FUNCTION_BLOCK FB_Cylinder IMPLEMENTS I_Cylinder
VAR_INPUT
	id	: INT;
END_VAR
VAR_OUTPUT
END_VAR
VAR
	bAtExtend 		AT %I*	: BOOL;
	bAtRetract 		AT %I*	: BOOL;
	bAtRetract_2	AT %I*	: BOOL;
	bMoveExtend 	AT %Q*	: BOOL;
	bMoveRetract 	AT %Q*	: BOOL;
END_VAR

PROPERTY bIsExtend : BOOL
GET
bIsExtend := bAtExtend;
END_GET
END_PROPERTY

PROPERTY bIsRetract : BOOL
GET
bIsRetract := bAtRetract;
END_GET
END_PROPERTY

METHOD Extend : BOOL
VAR_INPUT
END_VAR
bMoveExtend := TRUE;
bMoveRetract := FALSE;
END_METHOD

METHOD Retract : BOOL
VAR_INPUT
END_VAR
bMoveExtend := FALSE;
bMoveRetract := TRUE;
END_METHOD

END_FUNCTION_BLOCK

(* stored: Version 1.1.0.1, ProductVersion 3.1.4024.12
   POU FB_Cylinder: Id {ab010b65-5990-4cbd-8076-21ab8731ea05}, SpecialFunc None
   Property bIsExtend: Id {183076c0-a74e-46aa-8377-4ab639493447}
   Get Get: Id {bf6f37c2-9c1f-4bd4-af28-9ae7e5a181f6}
   Property bIsRetract: Id {f987a6d2-6fab-4f2f-89e8-c6c6c4438ea5}
   Get Get: Id {4e534881-8dc9-446b-a0fb-f9c80fcfa625}
   Method Extend: Id {9e3700c7-40fa-46ec-bca0-619165ac8f87}
   Method Retract: Id {05ea6731-f516-40c5-9773-eb913b2316a9} *)
